(* PLC project 117_1_V0.5.project, CODESYS CODESYS V3.5 SP17 Patch 3 *)
(* stored: creationDateTime 1970-01-01T00:00:00, modificationDateTime 2026-06-16T22:51:19.9979415 *)

FUNCTION_BLOCK StandLogic
  VAR_INPUT
    {attribute 'symbol' := 'none'}
    TimeManager : REFERENCE TO TimeManager;
    {attribute 'symbol' := 'none'}
    InputManager : REFERENCE TO InputManager;
    {attribute 'symbol' := 'none'}
    PIDController : REFERENCE TO BasicPIDController;
    {attribute 'symbol' := 'none'}
    ServoDriver : REFERENCE TO SM3ServoDriver;
    {attribute 'symbol' := 'none'}
    OutputManager : REFERENCE TO OutputManager;
  END_VAR
  VAR
    {attribute 'symbol' := 'none'}
    isError : BOOL := FALSE;
    {attribute 'symbol' := 'none'}
    isStateAxisOperational : BOOL := FALSE;
    {attribute 'symbol' := 'none'}
    isPowerStatus : BOOL := FALSE;
    {attribute 'symbol' := 'none'}
    isMoving : BOOL := FALSE;
    {attribute 'symbol' := 'none'}
    powerInclusionComplited : BOOL := FALSE;
    {attribute 'symbol' := 'none'}
    powerShutdownComplited : BOOL := FALSE;
    {attribute 'symbol' := 'none'}
    _controlMode : CONTROL_MODE := MANUAL;
    {attribute 'symbol' := 'none'}
    isExciterEnabled : BOOL := FALSE;
    {attribute 'symbol' := 'none'}
    isInputsReaded : BOOL;
    {attribute 'symbol' := 'none'}
    isForceRemoveLimitSwitchOn : BOOL;
    autoMoveStatus : AUTO_MOVE_STEPS := AWAIT;
    objectStatus : STATUS := NOT_COMMUNICATION;
    waitExciterOnTime : TIME := TIME#2s0ms;  (* Все что Время вкл/откл возбудителя *)
    waitExciterOffTime : TIME := TIME#2s0ms;
    cmdExciterOnOff : BOOL;  (* Команды Включение силовозбудителя *)
    cmdDisableExciter : BOOL;
    cmdPowerOn : BOOL;
    cmdPowerOff : BOOL;
    cmdErrorsReset : BOOL;
    cmdForwardJogging : BOOL;
    cmdBackwardJogging : BOOL;
    cmdChangeControlMode : BOOL;
    joggingVelocity : LREAL;  (* Ручное перемещение *)
    joggingAcceleration : LREAL;
    joggingDeceleration : LREAL;
    joggingJerk : LREAL;
    errorExciterEnableTime : BOOL;  (* Ошибки *)
    errorExciterDisableTime : BOOL;
    allErrors : ARRAY[0..15] OF BOOL;
    isInitialization : BOOL := TRUE;
    isInitialized : BOOL := FALSE;
    val : REAL;
    cc : INT;
    tenzaSensorDataArr : ARRAY[0..49] OF REAL;
    displacementSensorArr : ARRAY[0..49] OF REAL;
    nowSetpoint : REAL := 600;
    qq : BOOL;
    zz : BOOL;
    ExciterOn : SwitchingWithFeedbackControl;
    ExciterOff : SwitchingWithFeedbackControl;
    RemovingLimitSwitch : SwitchingWithFeedbackControl;
    pidStepKp : REAL;
    pidStepKi : REAL;
    pidStepKd : REAL;
    algSteps : UINT;
    stepFunction : UINT;
    diLiveCircuitsDC : BOOL;  (* Все нужные DI *)
    diFirstAlarmMushroom : BOOL;
    diSecondAlarmMushroom : BOOL;
    diLiveCircuitsAC : BOOL;
    diUpsDC_OK : BOOL;
    diUpsBattaryBad : BOOL;
    diUpsBattaryWork : BOOL;
    diUpperLimitSwitch : BOOL;
    diLowerLimitSwitch : BOOL;
    diRemovingLimitSwitch : BOOL;
    diExciter : BOOL;
    diLeftDoor : BOOL;
    diRightDoor : BOOL;
    doForcePowerLightColumn : BOOL;  (* Для поджига DO *)
    doForceRedLightColumn : BOOL;
    doForceGreenLightColumn : BOOL;
    doForceBuzzerLightColumn : BOOL;
    doForceExciter : BOOL;
    doForceRemoveLimitSwitch : BOOL;
    doStatePowerLightColumn : BOOL;  (* Состояние DO *)
    doStateRedLightColumn : BOOL;
    doStateGreenLightColumn : BOOL;
    doStateBuzzerLightColumn : BOOL;
    doStateExciter : BOOL;
    doStateRemoveLimitSwitch : BOOL;
  END_VAR

            // Чтение дискретных входов
isInputsReaded			:= _read_inputs();

// Проверка состояния силовозбудителя
isExciterEnabled		:= _check_exciter();

// Проверка состояния снятия с концевиков
isForceRemoveLimitSwitchOn := _check_removing_limit_switch();

// Проверка связи с драйвером
isStateAxisOperational	:= ServoDriver.get_axis_communication();
		
// Проверка наличия питания драйвера
isPowerStatus			:= ServoDriver.get_power_status();

IF NOT isInitialized THEN
	isInitialized := _init(TRUE);
ELSE
	// Включение и отключение дравера
	_driver_power(cmdPowerOn, cmdPowerOff);	
	
	// Режим управления
	CASE read_control_mode OF 
		MANUAL: //Ручное управление
			isMoving := _jogging(
							cmdForward 	 := cmdForwardJogging,
							cmdBackward  := cmdBackwardJogging,
							velocity	 := joggingVelocity,	
			         		acceleration := joggingAcceleration,	
			         		deceleration := joggingDeceleration,
			         		jerk		 := joggingJerk);	
							
		AUTO: // Автоматическое по алгоритму
			;
	END_CASE
	

END_IF
	














 
 IF cc >= 49 THEN
	cc := 0;
ELSE
	cc:= cc + 1;
END_IF

IF val  = 1000 THEN
	qq := TRUE;
	zz := FALSE;
ELSIF val = 0 THEN
	qq := FALSE;
	zz := TRUE;
END_IF

IF qq THEN 
		val := val - 1;
ELSIF zz THEN 
	val := val + 1;
END_IF


tenzaSensorDataArr[cc] := val;
displacementSensorArr[cc] := val + 100.0;
	

	
	//Сброс ошибок
	_reset_alarms(cmdErrorsReset);

	



	

	

	
	
	
	
	
// При аварии колонна подсвечивается красным и включается зуммер
_alarm_notification(FALSE);

// Запись статуса
objectStatus := _get_status();

// Запись выходов
_write_outputs();

          

METHOD _move_algorythm : BOOL
  VAR_INPUT
    enable : BOOL;
    kp : REAL;
    ki : REAL;
    kd : REAL;
    min_out : REAL;
    max_out : REAL;
    pv : REAL;
    sp : REAL;
    laststep : BOOL;
  END_VAR
                  IF enable THEN
	PIDController.Set_Configuration(
								Kp		:= kp,
								Ki		:= ki,
								Kd		:= kd,
								MinOut	:= min_out,
								MaxOut	:= max_out,
								Ts		:= TimeManager.get_interval_time_type_TIME(ms),
	);
															
PIDController.Enable();



PIDController.Reset();

PIDController.Get_Diagnostics();



// Управление скоростью
_move_algorythm := ServoDriver.start_follow_velocity(PIDController.xOutput);

ELSE
	PIDController.Disable();
	_move_algorythm := ServoDriver.stop_follow_velocity();
END_IF
                
END_METHOD

METHOD _get_status : STATUS
                  IF isError THEN
    _get_status := ERROR;
ELSIF NOT isStateAxisOperational THEN
    _get_status := NOT_COMMUNICATION;
ELSIF NOT isPowerStatus THEN
    _get_status := OFF;
ELSIF isMoving THEN
    _get_status := MOVING;
ELSE
    _get_status := READY;
END_IF
		

                
END_METHOD

METHOD _change_control_mode : CONTROL_MODE
  VAR_IN_OUT
    changeMode : BOOL;
  END_VAR
                  IF changeMode THEN
	IF isMoving THEN
		changeMode := FALSE;
	ELSE 
		IF (_controlMode = MANUAL) THEN
			_controlMode := AUTO;
			changeMode	:= FALSE;
		ELSIF (_controlMode = AUTO) THEN
			_controlMode := MANUAL;
			changeMode	:= FALSE;
		END_IF
	END_IF
END_IF

_change_control_mode := _controlMode;
                
END_METHOD

METHOD _jogging : BOOL
  VAR_INPUT
    cmdForward : BOOL;  (* Команда на прямое перемещение *)
    cmdBackward : BOOL;  (* Команда на обратное перемещение *)
    velocity : LREAL;  (* Скорость перемещения *)
    acceleration : LREAL;  (* Ускорение *)
    deceleration : LREAL;  (* Замедление *)
    jerk : LREAL;  (* Резкость ускорения *)
  END_VAR
                  
                
END_METHOD

METHOD _init : BOOL
  VAR_INPUT
    execute : BOOL;
    exciterEnable : BOOL := FALSE;
    LimitSwitch : BOOL := FALSE;
  END_VAR
  VAR
    vv : BYTE;
  END_VAR
                  

ServoDriver.set_power_on();
doForceExciter				:= TRUE;
doForceRemoveLimitSwitch	:= FALSE;


vv.0 := exciterEnable;

_init :=  isError;
                
END_METHOD

(* Поджигает светосигнальную колонну красным *)
METHOD _alarm_notification : BOOL
  VAR_INPUT
    alarm : BOOL := FALSE;
  END_VAR
                  IF alarm THEN 
	OutputManager.set_data(varName := outRedLightColumn,	enable := TRUE);
	OutputManager.set_data(varName := outBuzzerLightColumn, enable := TRUE);
ELSE
	OutputManager.set_data(varName := outRedLightColumn,	enable := FALSE);
	OutputManager.set_data(varName := outBuzzerLightColumn, enable := FALSE);
END_IF
                
END_METHOD

METHOD _read_inputs : BOOL
                  diLiveCircuitsDC		:= InputManager.get_discrete_data(inLiveCircuitsDC);
diFirstAlarmMushroom	:= InputManager.get_discrete_data(inFirstAlarmMushroom);
diSecondAlarmMushroom	:= InputManager.get_discrete_data(inSecondAlarmMushroom);
diLiveCircuitsAC		:= InputManager.get_discrete_data(inLiveCircuitsAC);
diUpsDC_OK				:= InputManager.get_discrete_data(inUpsDC_OK);
diUpsBattaryBad			:= InputManager.get_discrete_data(inUpsBattaryBad);
diUpsBattaryWork		:= InputManager.get_discrete_data(inUpsBattaryWork);
diUpperLimitSwitch		:= InputManager.get_discrete_data(inUpperLimitSwitch);
diLowerLimitSwitch		:= InputManager.get_discrete_data(inLowerLimitSwitch);
diRemovingLimitSwitch	:= InputManager.get_discrete_data(inRemovingLimitSwitch);
diExciter				:= InputManager.get_discrete_data(inExciter);
diLeftDoor				:= InputManager.get_discrete_data(inLeftDoor);
diRightDoor				:= InputManager.get_discrete_data(inRightDoor);

_read_inputs := TRUE;
                
END_METHOD

METHOD _collect_errors : BOOL
  VAR
    i : ERROR_INDEX;
    errors : WORD;
  END_VAR
                  

FOR i := communication TO lastIndex - 1 DO
    IF ServoDriver.get_axis_errors(i) THEN
        errors := errors OR SHL(WORD#1, i);
    ELSE
        errors := errors AND NOT SHL(WORD#1, i);
    END_IF
END_FOR

IF errors > 0 THEN
	objectStatus := ERROR;
END_IF
                
END_METHOD

(* Включение и отключение драйвера *)
METHOD _driver_power : BOOL
  VAR_IN_OUT
    PowerOnCmd : BOOL;  (* Команда на включение *)
    PowerOffCmd : BOOL;  (* Команда на отключение *)
  END_VAR
                  // Входные аргументы методов включения и отключения драйвера
// нужны для корретного завершения вызова методов.
// Т.к логика методов работает по шагам,
// на следующих циклах после начала выполнения метода,
// isPowerStatus сигнализирует о включенном питании,
// тем самым заставляя метод прервать выполнение логики

// Включение
IF PowerOnCmd THEN
	IF powerInclusionComplited := ServoDriver.set_power_on(isPowerStatus AND powerInclusionComplited) THEN
		powerInclusionComplited := FALSE;
		PowerOnCmd				:= FALSE;
	END_IF
	// Отключение
ELSIF PowerOffCmd THEN
	IF powerShutdownComplited := ServoDriver.set_power_off(NOT isPowerStatus AND powerShutdownComplited) THEN 
		powerShutdownComplited	:= FALSE;
		PowerOffCmd				:= FALSE;
	END_IF
END_IF
                
END_METHOD

METHOD _write_outputs : BOOL
                  doStatePowerLightColumn		:= OutputManager.set_data(outPowerLightColumn	, doForcePowerLightColumn);	 
doStateRedLightColumn 	 	:= OutputManager.set_data(outRedLightColumn		, doForceRedLightColumn); 	 
doStateGreenLightColumn		:= OutputManager.set_data(outGreenLightColumn	, doForceGreenLightColumn);	 
doStateBuzzerLightColumn	:= OutputManager.set_data(outBuzzerLightColumn	, doForceBuzzerLightColumn);
doStateExciter		   		:= OutputManager.set_data(outExciter			, doForceExciter);		 
doStateRemoveLimitSwitch	:= OutputManager.set_data(outRemoveLimitSwitch	, doForceRemoveLimitSwitch);
                
END_METHOD

METHOD _reset_alarms : BOOL
  VAR_INPUT
    ResetError : BOOL;
  END_VAR
                  IF ResetError THEN 
	IF ServoDriver.reset_errors() THEN 
	;
	END_IF
	cmdErrorsReset := FALSE;
END_IF
                
END_METHOD

METHOD _check_exciter : BOOL
                  _check_exciter := diExciter AND doStateExciter;

                
END_METHOD

METHOD _check_removing_limit_switch : BOOL
                  _check_removing_limit_switch := diRemovingLimitSwitch AND doStateRemoveLimitSwitch;

                
END_METHOD

PROPERTY read_control_mode : CONTROL_MODE
GET
                    
read_control_mode := _controlMode;
                  
END_GET
END_PROPERTY
END_FUNCTION_BLOCK
